PROGRAM POU
VAR
	Container_in_place : BOOL;
	Container_full : BOOL;
	Tank_empty_in : BOOL;
	Loading : BOOL;
	Unloading : BOOL;
	Start : BOOL;
	Stop : BOOL;
	Emergency : BOOL;
	
	Motor : BOOL;
	Valve : BOOL;
	Tank_empty_out : BOOL;
	counter: INT;
	R_TRIG_0: R_TRIG;
END_VAR

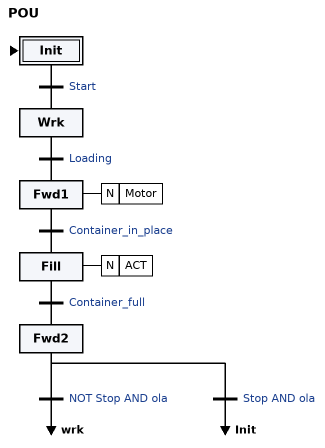
INITIAL_STEP Init:
END_STEP
TRANSITION FROM Init TO Wrk
    := Start;
END_TRANSITION
STEP Wrk:
END_STEP
TRANSITION FROM Wrk TO Fwd1
    := Loading;
END_TRANSITION
STEP Fwd1:
    Motor(N);
END_STEP
TRANSITION FROM Fwd1 TO Fill
    := Container_in_place;
END_TRANSITION
STEP Fill:
    ACT(N);
END_STEP
TRANSITION FROM Fill TO Fwd2
    := Container_full;
END_TRANSITION
STEP Fwd2:
END_STEP
TRANSITION FROM Fwd2 TO wrk
    := NOT Stop AND ola;
END_TRANSITION
TRANSITION FROM Fwd2 TO Init
    := Stop AND ola;
END_TRANSITION

ACTION ACT:
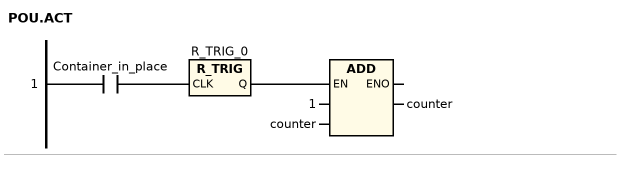
// NETWORK 1
R_TRIG_0(CLK := Container_in_place); // R_TRIG
IF R_TRIG_0.Q THEN counter := 1 + counter; END_IF
END_ACTION

TRANSITION ola:
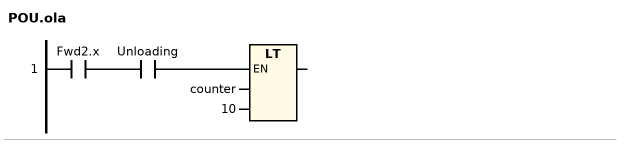
// NETWORK 1
(* Fwd2.x AND Unloading AND counter < 10; result not used *)
END_TRANSITION

END_PROGRAM

(* stored: Version 1.1.0.1, ProductVersion 3.1.4020.6
   POU POU: Id {2bab07bd-98e9-484f-9724-a0103e925e84}, SpecialFunc None
   Action ACT: Id {0c0a120e-0e60-434d-b7b6-8de5a90a011c}
   Transition ola: Id {b8729de7-90a3-4cf7-aa6f-95526c8c6aaa} *)
